{attribute 'GeneratedUsingTerminal: KL2032'}
{attribute addProperty BoxType "KL2032"}
{attribute addProperty Description ""}
{attribute addProperty Physics ""}
{attribute addProperty Id "Channel_1AT %Q*Channel_460B8C400Channel_2AT %Q*Channel_460B8C400"}
{attribute addProperty CRC "3701954066"}
{attribute addProperty Size "0"}
TYPE KL2032_DCA75612 :
STRUCT
	{attribute addProperty Name "Channel_1"}
	Channel_1 : Channel_460B8C40;
	{attribute addProperty Name "Channel_2"}
	Channel_2 : Channel_460B8C40;
END_STRUCT
END_TYPE

(* stored: Version 1.2.0.0, ProductVersion 3.1.4024.9
   DUT KL2032_DCA75612: Id {85057c16-2d7d-4cf5-899b-60ac6d55e02a} *)
